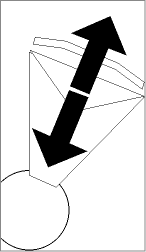
VISUALIZATION VISU_CoverPanelDrawing  // 146x252
VAR_IN_OUT
    coverPanelConfig : CoverPanelConfig;
	coverPanel : CoverPanel;
	widget : CoverPanelWidget;
END_VAR
    Ellipse (-11,170 80x80), invisible if: TRUE
    Polygon (29,175) (56,187) (144,97) (29,52), invisible if: NOT coverPanel.statuses.apertureStatus.closed, colour variable: widget.actualStatus.color.bg
        p2858320360: coverPanelConfig.offset
    Polygon (66,101) (66,101) (84,109) (144,96) (144,96) (30,50), invisible if: NOT coverPanel.statuses.apertureStatus.partiallyOpen, colour variable: widget.actualStatus.color.bg
        p2858320360: coverPanelConfig.offset
    Polygon (144,82) (118,63) (66,41) (35,37) (33,44) (63,48) (115,69) (142,89), invisible if: NOT coverPanel.statuses.apertureStatus.open, colour variable: widget.actualStatus.color.bg
        p2858320360: coverPanelConfig.offset
    Polygon (89,94) (70,86) (89,40) (71,33) (110,16) (126,55) (108,48), invisible if: NOT coverPanel.statuses.openingStatus.opening
        p2858320360: coverPanelConfig.offset
    Polygon (69,90) (88,97) (69,143) (87,151) (48,167) (32,128) (50,136), invisible if: NOT coverPanel.statuses.openingStatus.closing
        p2858320360: coverPanelConfig.offset
END_VISUALIZATION

(* stored: Version 1.1.0.1, ProductVersion 3.1.0.36
   Visu VISU_CoverPanelDrawing: Id {0d8cebce-1bbc-4d99-929e-3616e097278e} *)
